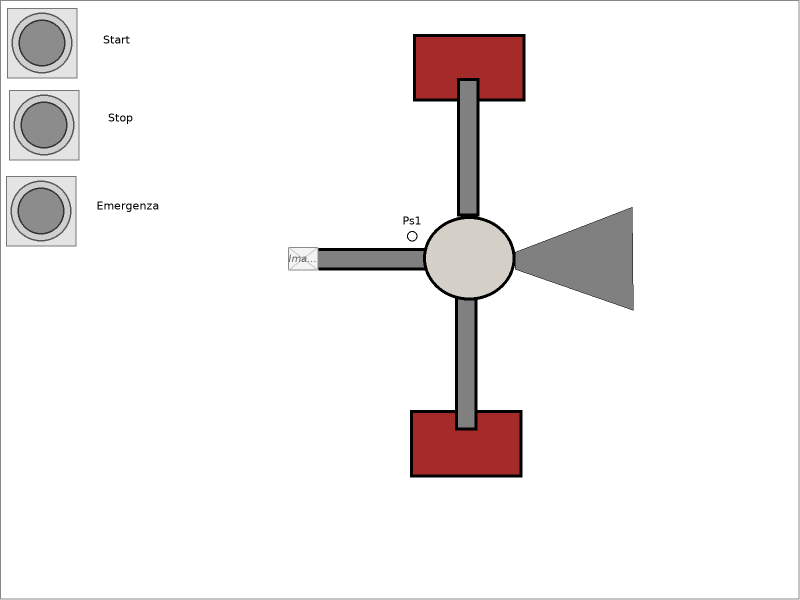
VISUALIZATION Visualization  // 800x600
    Rectangle (473,-103 67x112), angle 270
    Rectangle (470,273 67x112), angle 270
    Rectangle (856,994 145x265), angle 270
    PushSwitch (7,8 70x70), behaviour: TAP, style: Switch-PushSwitch-Gray
    Label (89,25 55x30), "Start"
    PushSwitch (9,90 70x70), behaviour: TAP, style: Switch-PushSwitch-Gray
    Label (88,103 65x30), "Stop"
    PushSwitch (6,176 70x70), behaviour: TAP, style: Switch-PushSwitch-Gray
    Label (83,191 90x30), "Emergenza"
    Rectangle (289,248 138x22)
    Rectangle (304,201 138x22), angle 90
    Rectangle (302,415 138x22), angle 90
    Ellipse (423,216 92x84)
    Polygon (515,252) (557,236) (632,207) (633,310) (515,269)
    Image (288,247 30x23), image: ImagePool.ham
    Ellipse (407,231 10x10), colour toggle: GVL.bPs1
    Label (388,215 48x12), "Ps1"
END_VISUALIZATION

(* stored: Version 1.1.0.1, ProductVersion 3.1.4024.12
   Visu Visualization: Id {e3399594-b7fd-4589-9a49-3967da9e8e84} *)
